Fanuc KAREL source: IO0089.KL

-- PROVISIONAL review KL for V940-1; original PC SHA256 db057c53e38fffa3771c065aa8220c03fc9af92ac3f5f3da549e268f704d9ca5
-- Incomplete behavior may be omitted. Consult companion uncertainty JSON. Do not deploy.
PROGRAM IO0089
%NOLOCKGROUP
-- UNRESOLVED_LOCAL_POOL 5 cells at code offset 13; source declarations unknown
-- DIRECT_LOCAL_WORD_ACCESS alone does not prove INTEGER, REAL, or BOOLEAN
BEGIN
  -- V9_EXPOSED_INDEXED_TABLE_HINT layout=0001; 1 counted words exposed once; source arms/runtime held
  -- V9_ZERO_GLOBAL_LAYOUT_HINT count-one $GROUP table, zero relocation slots, two routine descriptors; executable preamble and source held
  -- V9_ANALOG_RDI_SIGNAL_HINT AOUT condition I_plus_1
  -- UNRESOLVED_PC offsets 0-18; opcodes 2B,2C,7B
  -- UNRESOLVED_PC offsets 23-30; opcodes 9D,23
  -- UNRESOLVED_PC offsets 35-49; opcodes 2E,22,9D,33,35
  -- UNRESOLVED_PC offsets 54-61; opcodes 9D,23
  -- UNRESOLVED_PC offsets 66-77; opcodes 2E,23
  -- UNRESOLVED_PC offsets 82-99; opcodes 21,9D,52,19,9C,5B,79
  -- UNRESOLVED_PC offsets 104-118; opcodes 21,9D,52,23
  -- UNRESOLVED_PC offsets 128-132; opcodes 7F
  -- UNRESOLVED_PC offsets 137-141; opcodes 27,AA
  -- UNRESOLVED_PC offsets 146-150; opcodes 7F
END IO0089
